(* IEC 61131-3 sources: programs/VI-54/VI-54_20171205/VI-54_20171205/Stations/Screen/LseClass170718/Class/ReadValue, 1 file *)

(* ---- ReadValue.st ---- *)
(*!
<Class
	Name               = "ReadValue"
	Revision           = "1.1"
	RealtimeTask       = "false"
	CyclicTask         = "false"
	BackgroundTask     = "false"
	Sigmatek           = "false"
	OSInterface        = "false"
	HighPriority       = "false"
	Automatic          = "false"
	UpdateMode         = "Prescan"
	SharedCommandTable = "true"
	Objectsize         = "(588,120)"
	Comment            = "Diese Klasse dient in Verbindung mit der Klasse SynchRdWr zum Versenden bzw. Empfangen von 4 Byte Werten einer verbundenen Steuerung.">
	<Channels>
		<Server Name="ClassSvr" Visualized="false" Initialize="false" WriteProtected="true" Retentive="false" Comment="READY.. Registration at manager class (TCPComReceiveData) was successful&#13;&#10;ERROR.. Registration failed"/>
		<Server Name="RxServer" Visualized="false" Initialize="false" WriteProtected="true" Retentive="false" Comment="This server shows the last received value"/>
		<Client Name="coSystemLogging" Required="false" Internal="false" Comment="object channel to SystemLogging (optional)"/>
		<Client Name="coTCPComReceive" Required="true" Internal="false" Comment="Object channel to TCPComReceiveData"/>
		<Client Name="ID" Required="true" Internal="false" Comment="ID number which must be unique for each object. It also must be the same number like the ID of the sending object, so that this class receives its data."/>
		<Client Name="RxClient" Required="false" Internal="false" Comment="When receiving data, the received value will be set on this client, and written to the connected server."/>
	</Channels>
	<RevDoku>
		<Owner Company="Sigmatek"/>
		<Dokumentation Revision="1.1" Date="2015-09-29" Author="BraLis" Company="Sigmatek" Description="insert the method SystemLogging::LogEventText instead of TRACE-Messages"/>
		<Dokumentation Revision="1.0" Date="2015-03-31" Company="Sigmatek"/>
	</RevDoku>
</Class>
*)
ReadValue : CLASS
	TYPE
#pragma pack(push, 1)
	  RdData : STRUCT
	    udID : UDINT;
	    dValue : DINT;
	  END_STRUCT;
#pragma pack(pop)
	END_TYPE
  //Servers:
	ClassSvr 	: SvrChCmd_iprStates;
	RxServer 	: SvrCh_DINT;
  //Clients:
	coTCPComReceive 	: CltChCmd_TCPComReceiveData;
	ID 	: CltCh_UDINT;
	RxClient 	: CltCh_DINT;
	coSystemLogging 	: CltChCmd_SystemLogging;
  //Variables:
		usInitRun 	: USINT;
		aRdData 	: RdData;
  //Functions:

	FUNCTION VIRTUAL GLOBAL Init;
				//! <Function Comment="When receiving data, this method will be called by the class TCPComReceiveData. It sets the client RxClient and the server RxServer to the received value." Name="SetData"/>
	FUNCTION VIRTUAL GLOBAL SetData
		VAR_INPUT
			pValue 	: ^void;			//! <Variable Comment="Pointer to the received data" Name="SetData.pValue"/>
			udSize 	: UDINT;			//! <Variable Comment="Size of the received data" Name="SetData.udSize"/>
		END_VAR
		VAR_OUTPUT
			bSuccessful 	: BOOL;			//! <Variable Comment="TRUE..  Successfully received the data&#13;&#10;FALSE.. Wrong size of the received data" Name="SetData.bSuccessful"/>
		END_VAR;
  //Tables:
	FUNCTION @STD
		VAR_OUTPUT
			ret_code	: CONFSTATES;
		END_VAR;
	FUNCTION GLOBAL TAB @CT_;
END_CLASS;

#pragma usingLtd SystemLogging
#pragma usingLtd TCPComReceiveData

FUNCTION VIRTUAL GLOBAL ReadValue::Init

  // erster Init-Durchlauf
  //------------------------------------------------------
  if usInitRun = 0 then

    // ID-Nummer lesen
    ID := ID.Read();

    // Anmelden an Manager Klasse
    if coTCPComReceive.LoginObject(udID  := ID,
                                pThis := this) = true then
      ClassSvr := READY;
    else
      if (IsClientConnected(input:=#coSystemLogging)) then
        coSystemLogging.LogEventText("WriteValue::Init(): Anmelden an Manager Klasse fehlgeschlagen");
      end_if;
      ClassSvr := ERROR;
    end_if;

  end_if;

  // Init-Durchlauf zählen
  usInitRun += 1;

END_FUNCTION

FUNCTION VIRTUAL GLOBAL ReadValue::SetData
	VAR_INPUT
		pValue 	: ^void;
		udSize 	: UDINT;
	END_VAR
	VAR_OUTPUT
		bSuccessful 	: BOOL;
	END_VAR

  if udSize = sizeof(RdData) then

    aRdData := pValue^$RdData;

    // Wert auf Client setzen und schreiben
    RxClient := aRdData.dValue;
    RxClient.Write(RxClient);

    // Wert auf Server setzen
    RxServer := aRdData.dValue;

    // Rückgabewert setzen, alles erfolgreich
    bSuccessful := true;

  else

    bSuccessful := false;

  end_if;

END_FUNCTION
